TYPE ST_EM_Lift_Hmi :
STRUCT
	fbMotorLift : HMI_CM_ServoAX8000;
END_STRUCT
END_TYPE

(* stored: Version 1.1.0.1, ProductVersion 3.1.4026.13
   DUT ST_EM_Lift_Hmi: Id {0ad72c98-9a1e-44d6-8240-055cab49aae8} *)
